{attribute 'GeneratedUsingTerminal: EK1100-0000-0018'}
{attribute addProperty BoxType "EK1100-0000-0018"}
{attribute addProperty Id "R1_A4_X2_A2_EK1122R1_A4_X2_A2_EK1122_39ABCC27250R1_A4_X2_IA1_EL1809EL1809_32157CFD20R1_A4_X2_IA2_EL1809EL1809_32157CFD20R1_A4_X2_IA3_EL1809EL1809_32157CFD20R1_A4_X2_IA4_EL1809EL1809_32157CFD20R1_A4_X2_IA5_EL1809EL1809_32157CFD20R1_A4_X2_QA1_EL2809EL2809_2B6483BD19R1_A4_X2_QA2_EL2809EL2809_2B6483BD19R1_A4_X2_QA3_EL2809EL2809_2B6483BD19R1_A4_X2_EndTerminal_EL9010EL9010_D29C20850"}
{attribute addProperty CRC "1868542906"}
{attribute addProperty Size "407"}
{attribute addProperty Name "R1_A4_X2 (EK1100)"}
TYPE R1_A4_X2_EK1100_6F5FB3BA EXTENDS EK1100_1FC0878B :
STRUCT
	{attribute addProperty Name "R1_A4_X2_A2 (EK1122)"}
	{attribute addProperty PreviousPort "R1_A4_X2 (EK1100) : B"}
	R1_A4_X2_A2_EK1122 : R1_A4_X2_A2_EK1122_39ABCC27;
	{attribute addProperty Name "R1_A4_X2_IA1 (EL1809)"}
	{attribute addProperty PreviousPort "R1_A4_X2_A2 (EK1122) : C"}
	R1_A4_X2_IA1_EL1809 : EL1809_32157CFD;
	{attribute addProperty Name "R1_A4_X2_IA2 (EL1809)"}
	{attribute addProperty PreviousPort "R1_A4_X2_IA1 (EL1809) : B"}
	R1_A4_X2_IA2_EL1809 : EL1809_32157CFD;
	{attribute addProperty Name "R1_A4_X2_IA3 (EL1809)"}
	{attribute addProperty PreviousPort "R1_A4_X2_IA2 (EL1809) : B"}
	R1_A4_X2_IA3_EL1809 : EL1809_32157CFD;
	{attribute addProperty Name "R1_A4_X2_IA4 (EL1809)"}
	{attribute addProperty PreviousPort "R1_A4_X2_IA3 (EL1809) : B"}
	R1_A4_X2_IA4_EL1809 : EL1809_32157CFD;
	{attribute addProperty Name "R1_A4_X2_IA5 (EL1809)"}
	{attribute addProperty PreviousPort "R1_A4_X2_IA4 (EL1809) : B"}
	R1_A4_X2_IA5_EL1809 : EL1809_32157CFD;
	{attribute addProperty Name "R1_A4_X2_QA1 (EL2809)"}
	{attribute addProperty PreviousPort "R1_A4_X2_IA5 (EL1809) : B"}
	R1_A4_X2_QA1_EL2809 : EL2809_2B6483BD;
	{attribute addProperty Name "R1_A4_X2_QA2 (EL2809)"}
	{attribute addProperty PreviousPort "R1_A4_X2_QA1 (EL2809) : B"}
	R1_A4_X2_QA2_EL2809 : EL2809_2B6483BD;
	{attribute addProperty Name "R1_A4_X2_QA3 (EL2809)"}
	{attribute addProperty PreviousPort "R1_A4_X2_QA2 (EL2809) : B"}
	R1_A4_X2_QA3_EL2809 : EL2809_2B6483BD;
	{attribute addProperty Name "R1_A4_X2_EndTerminal (EL9010)"}
	{attribute addProperty PreviousPort "R1_A4_X2_QA3 (EL2809) : B"}
	R1_A4_X2_EndTerminal_EL9010 : EL9010_D29C2085;
END_STRUCT
END_TYPE

(* stored: Version 1.2.0.0, ProductVersion 3.1.4024.11
   DUT R1_A4_X2_EK1100_6F5FB3BA: Id {4f99f4a5-97cf-015d-2a47-0d43e8456030} *)
